// TIA Portal project "1905391_000_002" (V16)

(* hardware
DEVICE "S7-1200 station_1"  S7-1200 Station
   slot 0: "Rack_0"  S7-1200 Rack  Rack  V1.0
   slot 1: "PLC_1"  CPU 1211C DC/DC/DC  6ES7 211-1AE40-0XB0  V4.4
DEVICE "HMI_1"  TP900 Comfort
   slot 0: "HMI_1"  TP900 Comfort  6AV2 124-0JC01-0AX0  16.0.0.0
   slot 1: "HMI_RT_1"  TP900 Comfort  6AV2 124-0JC01-0AX0  16.0.0.0
   slot 5: "HMI_1.IE_CP_1"  PROFINET Interface  16.0.0.0
      slot 1: "PROFINET Interface_1"  PROFINET Interface
         slot 1: "Port_1"  Port
         slot 2: "Port_2"  Port
   slot 7: "HMI_1.MPI/DP_CP_1"  MPI/DP Interface  16.0.0.0
*)

// ===== PLC "PLC_1"  CPU 1211C DC/DC/DC =====

VAR_GLOBAL   // PLC tag table "Default tag table"
   "System_Byte" AT %MB1 : Byte;
   "FirstScan" AT %M1.0 : Bool;
   "DiagStatusUpdate" AT %M1.1 : Bool;
   "AlwaysTRUE" AT %M1.2 : Bool;
   "AlwaysFALSE" AT %M1.3 : Bool;
   "Clock_Byte" AT %MB0 : Byte;
   "Clock_10Hz" AT %M0.0 : Bool;
   "Clock_5Hz" AT %M0.1 : Bool;
   "Clock_2.5Hz" AT %M0.2 : Bool;
   "Clock_2Hz" AT %M0.3 : Bool;
   "Clock_1.25Hz" AT %M0.4 : Bool;
   "Clock_1Hz" AT %M0.5 : Bool;
   "Clock_0.625Hz" AT %M0.6 : Bool;
   "Clock_0.5Hz" AT %M0.7 : Bool;
END_VAR

VAR_GLOBAL CONSTANT   // PLC tag table "Default tag table"
   "STRING_LENGTH" : Int := 20;
   "ADP_PARAMETER_LENGTH" : Int := 5;
END_VAR

TYPE "Database.UDT"
   STRUCT
      elements : "Elements.Data.UDT";
      wires : "Wires.Data.UDT";
   END_STRUCT;
END_TYPE

TYPE "Row.(IOF.String_IOF.String).UDT"
   STRUCT
      cell_00 : "IO_Field.String.UDT";
      cell_01 : "IO_Field.String.UDT";
   END_STRUCT;
END_TYPE

TYPE "IO_Field.String.UDT"
   STRUCT
      animation : Int;
      enable : Bool;
      input_finished : Bool;
      visible : Bool;
      value : String["STRING_LENGTH"];
   END_STRUCT;
END_TYPE

TYPE "HMI_Interface.UDT"
   STRUCT
      elements : "Elements.HMI.UDT";
      wires : "Wires.HMI.UDT";
   END_STRUCT;
END_TYPE

TYPE "LED_Interface.UDT"
   STRUCT
      elements : "Elements.LED.UDT";
      wires : "Wires.LED.UDT";
   END_STRUCT;
END_TYPE

TYPE "Row.(IOF.String_IOF.Real).UDT"
   STRUCT
      cell_00 : "IO_Field.String.UDT";
      cell_01 : "IO_Field.Real.UDT";
   END_STRUCT;
END_TYPE

TYPE "IO_Field.Real.UDT"
   STRUCT
      animation : Int;
      enable : Bool;
      input_finished : Bool;
      visible : Bool;
      value : Real;
   END_STRUCT;
END_TYPE

// folder: ADP Data

TYPE "ADP.Row.2_Cells.UDT"
   STRUCT
      me : Array[0..1] of "ADP.Cell.UDT";
   END_STRUCT;
END_TYPE

TYPE "ADP.Cell.UDT"
   STRUCT
      color : String["ADP_PARAMETER_LENGTH"];
      flashing : String["ADP_PARAMETER_LENGTH"];
      h_align : String["ADP_PARAMETER_LENGTH"];
      lince_control : String["ADP_PARAMETER_LENGTH"];
      scroll_speed : String["ADP_PARAMETER_LENGTH"];
      size_and_face : String["ADP_PARAMETER_LENGTH"];
      v_align : String["ADP_PARAMETER_LENGTH"];
      value : String["STRING_LENGTH"];
   END_STRUCT;
END_TYPE

TYPE "ADP.Message_Buffer.UDT"
   STRUCT
      me : Array[0..999] of Byte;
   END_STRUCT;
END_TYPE

TYPE "ADP.Decoded.UDT"
   STRUCT
      color : "ADP.Decoded.Color.UDT";
      flash : "ADP.Decoded.Flash.UDT";
      horizontal_alignment : "ADP.Decoded.Horizontal_Alignment.UDT";
      line_control : "ADP.Decoded.Line_Control.UDT";
      scroll_speed : "ADP.Decoded.Scroll_Speed.UDT";
      size_and_face : "ADP.Decoded.Size_and_Face.UDT";
      vertical_alignment : "ADP.Decoded.Vertical_Alignment.UDT";
   END_STRUCT;
END_TYPE

TYPE "ADP.Decoded.Color.UDT"
   STRUCT
      black : String[8] := 'black';
      blue : String[8] := 'blue';
      green : String[8] := 'green';
      mix_1 : String[8] := 'mix 1';
      mix_2 : String[8] := 'mix 2';
      mix_3 : String[8] := 'mix 3';
      mix_4 : String[8] := 'mix 4';
      red : String[8] := 'red';
      white : String[8] := 'white';
      yellow : String[8] := 'yellow';
   END_STRUCT;
END_TYPE

TYPE "ADP.Decoded.Flash.UDT"
   STRUCT
      off : String[8] := 'off';
      on : String[8] := 'on';
   END_STRUCT;
END_TYPE

TYPE "ADP.Decoded.Horizontal_Alignment.UDT"
   STRUCT
      center : String[8] := 'center';
      left : String[8] := 'left';
      right : String[8] := 'right';
   END_STRUCT;
END_TYPE

TYPE "ADP.Encoded.UDT"
VERSION : 0.1
   STRUCT
      file_system : "ADP.Encoded.File_System.UDT";
      formatting : "ADP.Encoded.Formatting.UDT";
   END_STRUCT;
END_TYPE

TYPE "ADP.Message_Formats.Encoded.UDT"
   STRUCT
      color : String [5];
      flash : String [5];
      scroll_speed : String [5];
      size_and_face : String [5];
      vertical_alignment : String [5];
      horizontal_alignment : String [5];
   END_STRUCT;
END_TYPE

TYPE "ADP.Message_Formats.Decoded.UDT"
   STRUCT
      color : String [20];
      flash : String [20];
      scroll_speed : String [20];
      size_and_face : String [20];
      vertical_alignment : String [20];
      horizontal_alignment : String [20];
   END_STRUCT;
END_TYPE

TYPE "ADP.Decoded.Scroll_Speed.UDT"
   STRUCT
      slowest : String[9] := 'slowest';
      slow : String[9] := 'slow';
      normal : String[9] := 'normal';
      fast : String[9] := 'fast';
      fastest : String[9] := 'fastest';
   END_STRUCT;
END_TYPE

TYPE "ADP.Decoded.Size_and_Face.UDT"
   STRUCT
      bold_5 : String[11] := 'bold 5';
      bold_11 : String[11] := 'bold 11';
      bold_14 : String[11] := 'bold 14';
      bold_15 : String[11] := 'bold 15';
      bold_16 : String[11] := 'bold 16';
      bold_22 : String[11] := 'bold 22';
      bold_30 : String[11] := 'bold 30';
      bold_32 : String[11] := 'bold 32';
      bold_40 : String[11] := 'bold 40';
      normal_5 : String[11] := 'normal 5';
      normal_7 : String[11] := 'normal 7';
      normal_9 : String[11] := 'normal 9';
      normal_11 : String[11] := 'normal 11';
      normal_14 : String[11] := 'normal 14';
      normal_15 : String[11] := 'normal 15';
      normal_16 : String[11] := 'normal 16';
      normal_22 : String[11] := 'normal 22';
      normal_24 : String[11] := 'normal 24';
      normal_30 : String[11] := 'normal 30';
      normal_32 : String[11] := 'normal 32';
      normal_40 : String[11] := 'normal 40';
   END_STRUCT;
END_TYPE

TYPE "ADP.Decoded.Vertical_Alignment.UDT"
   STRUCT
      bottom_hold : String[15] := 'bottom hold';
      fill_hold : String[15] := 'fill hold';
      middle_hold : String[15] := 'middle hold';
      top_hold : String[15] := 'top hold';
      bottom_scroll : String[15] := 'bottom scroll';
      fill_scroll : String[15] := 'fill scroll';
      middle_scroll : String[15] := 'middle scroll';
      top_scroll : String[15] := 'top scroll';
   END_STRUCT;
END_TYPE

TYPE "ADP.Encoded.File_System.UDT"
   STRUCT
      "00 Start of Header" : String[5] := '$01';
      "01 Address" : String[5] := 'Z00';
      "02 Start of Text" : String[5] := '$02';
      "03 Command & File" : String[5] := 'AA';
      "04 END" : String[5] := '$04';
   END_STRUCT;
END_TYPE

TYPE "ADP.Encoded.Formatting.UDT"
   STRUCT
      color : "ADP.Encoded.Formatting.Color.UDT";
      flashing : "ADP.Encoded.Formatting.Flashing.UDT";
      horizontal_alignment : "ADP.Encoded.Formatting.Horizonta_Alignment.UDT";
      line_control : "ADP.Encoded.Formatting.Line_Control.UDT";
      scroll_speed : "ADP.Encoded.Formatting.Scroll_Speed.UDT";
      size_and_face : "ADP.Encoded.Formatting.Size_and_Face.UDT";
      vertical_alignment : "ADP.Encoded.Formatting.Vertical_Alignment.UDT";
   END_STRUCT;
END_TYPE

TYPE "ADP.Encoded.Formatting.Color.UDT"
   STRUCT
      black : String[5] := '$1C0';
      blue : String[5] := '$1C8';
      green : String[5] := '$1C2';
      mix_1 : String[5] := '$1C4';
      mix_2 : String[5] := '$1C5';
      mix_3 : String[5] := '$1C6';
      mix_4 : String[5] := '$1CY';
      red : String[5] := '$1C1';
      white : String[5] := '$1C9';
      yellow : String[5] := '$1C3';
   END_STRUCT;
END_TYPE

TYPE "ADP.Encoded.Formatting.Flashing.UDT"
   STRUCT
      off : String[5] := '$070';
      on : String[5] := '$071';
   END_STRUCT;
END_TYPE

TYPE "ADP.Encoded.Formatting.Size_and_Face.UDT"
   STRUCT
      bold_5 : String[5] := '$1AG';
      bold_11 : String[5] := '$1AH';
      bold_14 : String[5] := '$1A5';
      bold_15 : String[5] := '$1A6';
      bold_16 : String[5] := '$1A7';
      bold_22 : String[5] := '$1AC';
      bold_30 : String[5] := '$1AI';
      bold_32 : String[5] := '$1AJ';
      bold_40 : String[5] := '$1AK';
      normal_5 : String[5] := '$1A0';
      normal_7 : String[5] := '$1A1';
      normal_9 : String[5] := '$1A8';
      normal_11 : String[5] := '$1A9';
      normal_14 : String[5] := '$1A2';
      normal_15 : String[5] := '$1A3';
      normal_16 : String[5] := '$1A4';
      normal_22 : String[5] := '$1AA';
      normal_24 : String[5] := '$1AB';
      normal_30 : String[5] := '$1AD';
      normal_32 : String[5] := '$1AE';
      normal_40 : String[5] := '$1AF';
   END_STRUCT;
END_TYPE

TYPE "ADP.Encoded.Formatting.Horizonta_Alignment.UDT"
   STRUCT
      center : String[5] := '$L1';
      left : String[5] := '$L0';
      right : String[5] := '$L2';
   END_STRUCT;
END_TYPE

TYPE "ADP.Encoded.Formatting.Vertical_Alignment.UDT"
   STRUCT
      middle_hold : String[5] := '$1B b';
      fill_hold : String[5] := '$1B"b';
      bottom_hold : String[5] := '$1B&b';
      top_hold : String[5] := '$1B0b';
      bottom_scroll : String[5] := '$1B a';
      fill_scroll : String[5] := '$1B"a';
      middle_scroll : String[5] := '$1B&a';
      top_scroll : String[5] := '$1B0a';
   END_STRUCT;
END_TYPE

TYPE "ADP.Encoded.Formatting.Scroll_Speed.UDT"
   STRUCT
      slowest : String[5] := '$15';
      slow : String[5] := '$16';
      normal : String[5] := '$17';
      fast : String[5] := '$18';
      fastest : String[5] := '$19';
   END_STRUCT;
END_TYPE

TYPE "ADP.Encoded.Formatting.Line_Control.UDT"
   STRUCT
      new_line : String[5] := '$R';
      word_wrap : String[5] := '';
   END_STRUCT;
END_TYPE

TYPE "ADP.Decoded.Line_Control.UDT"
   STRUCT
      new_line : String[9] := 'new line';
      word_wrap : String[9] := 'word wrap';
   END_STRUCT;
END_TYPE

// folder: Element Data

TYPE "Elements.HMI.UDT"
   STRUCT
      chromium : "Row.(IOF.String_IOF.Real).UDT";
      custom : "Row.(IOF.String_IOF.Real).UDT";
      header : "Row.(IOF.String_IOF.String).UDT";
      heat : "Row.(IOF.String_IOF.Real).UDT";
      manganese : "Row.(IOF.String_IOF.Real).UDT";
      molybdenum : "Row.(IOF.String_IOF.Real).UDT";
      nickel : "Row.(IOF.String_IOF.Real).UDT";
      silicon : "Row.(IOF.String_IOF.Real).UDT";
      vanadium : "Row.(IOF.String_IOF.Real).UDT";
   END_STRUCT;
   // header.cell_00.value := 'Material';
   // header.cell_01.value := 'Bags';
END_TYPE

TYPE "Elements.Data.UDT"
   STRUCT
      chromium : Real;
      custom : Real;
      heat : Real;
      manganese : Real;
      molybdenum : Real;
      nickel : Real;
      silicon : Real;
      vanadium : Real;
   END_STRUCT;
END_TYPE

TYPE "Elements.LED.UDT"
   STRUCT
      chromium : "ADP.Row.2_Cells.UDT";
      custom : "ADP.Row.2_Cells.UDT";
      header : "ADP.Row.2_Cells.UDT";
      heat : "ADP.Row.2_Cells.UDT";
      manganese : "ADP.Row.2_Cells.UDT";
      molybdenum : "ADP.Row.2_Cells.UDT";
      nickel : "ADP.Row.2_Cells.UDT";
      silicon : "ADP.Row.2_Cells.UDT";
      vanadium : "ADP.Row.2_Cells.UDT";
   END_STRUCT;
   // chromium.me[0].value := 'chromium';
   // heat.me[0].value := 'heat';
   // manganese.me[0].value := 'manganese';
   // molybdenum.me[0].value := 'molybdenum';
   // nickel.me[0].value := 'nickel';
   // silicon.me[0].value := 'silicon';
   // vanadium.me[0].value := 'vanadium';
   // custom.me[0].value := 'Custom';
   // header.me[0].value := 'Material';
   // header.me[1].value := 'Bags';
END_TYPE

// folder: Wire Data

TYPE "Wires.Data.UDT"
   STRUCT
      aluminum : Real;
      calcium_silicon : Real;
      carbon : Real;
      custom : Real;
      heat : Real;
      sulfur : Real;
   END_STRUCT;
END_TYPE

TYPE "Wires.LED.UDT"
   STRUCT
      aluminum : "ADP.Row.2_Cells.UDT";
      calcium_silicon : "ADP.Row.2_Cells.UDT";
      carbon : "ADP.Row.2_Cells.UDT";
      custom : "ADP.Row.2_Cells.UDT";
      heat : "ADP.Row.2_Cells.UDT";
      sulfur : "ADP.Row.2_Cells.UDT";
   END_STRUCT;
   // aluminum.me[0].value := 'AL Wire';
   // calcium_silicon.me[0].value := 'Cal/Sil Wire';
   // carbon.me[0].value := 'Carbon Wire';
   // heat.me[0].value := 'HEAT';
   // sulfur.me[0].value := 'Sulfur Wire';
   // custom.me[0].value := 'Custom';
END_TYPE

TYPE "Wires.HMI.UDT"
   STRUCT
      aluminum : "Row.(IOF.String_IOF.Real).UDT";
      calcium_silicon : "Row.(IOF.String_IOF.Real).UDT";
      carbon : "Row.(IOF.String_IOF.Real).UDT";
      custom : "Row.(IOF.String_IOF.Real).UDT";
      header : "Row.(IOF.String_IOF.String).UDT";
      heat : "Row.(IOF.String_IOF.Real).UDT";
      sulfur : "Row.(IOF.String_IOF.Real).UDT";
   END_STRUCT;
   // header.cell_00.value := 'Material';
   // header.cell_01.value := 'Feet';
END_TYPE

// folder: data

DATA_BLOCK "Database.Data"   // DB1
{ S7_Optimized_Access := 'TRUE' }
VERSION : 0.1
BEGIN
END_DATA_BLOCK

// folder: display/HMI

DATA_BLOCK "HMI_Interface.Data"   // DB2
{ S7_Optimized_Access := 'TRUE' }
VERSION : 0.1
BEGIN
END_DATA_BLOCK

// folder: display/LED

DATA_BLOCK "LED_Interface.Data"   // DB3
{ S7_Optimized_Access := 'TRUE' }
VERSION : 0.1
BEGIN
END_DATA_BLOCK

// folder: (top level)

FUNCTION "Strip_Sign" : String   // FC20, SCL
{ S7_Optimized_Access := 'TRUE' }
VERSION : 0.1
   VAR_INPUT
      "string" : String;
   END_VAR
   VAR_TEMP
      Length : Int;
      "String Box" : String;
      "Test Character" : String;
   END_VAR
   VAR CONSTANT
      "+" : Char := '+';
      "-" : Char := '-';
   END_VAR
BEGIN
   #"String Box" := #string;
   #"Test Character" := LEFT_STRING(IN := #"String Box",
                                    L := 1);
   IF #"Test Character" = #"+" OR #"Test Character" = #"-" THEN
       #Length := LEN(#"String Box");
       #"String Box" := RIGHT_STRING(IN := #"String Box", L := #Length - 1);

   END_IF;
   #"Strip Sign" := #"String Box";
END_FUNCTION

FUNCTION "Trim" : String   // FC21, SCL
{ S7_Optimized_Access := 'TRUE' }
AUTHOR : Machado
FAMILY : String
VERSION : 1.0
// removes leading and trailing whitespace from input string
   VAR_INPUT
      "string" : String;
   END_VAR
   VAR_TEMP
      ret : String;
   END_VAR
   VAR CONSTANT
      space : String := ' ';
   END_VAR
BEGIN
   #ret := #string;
   WHILE LEFT(IN := #ret, L := 1) = #space DO
       #ret := RIGHT(IN := #ret, L := LEN(#ret) - 1);
   END_WHILE;
   WHILE RIGHT(IN := #ret, L := 1) = #space DO
       #ret := LEFT(IN := #ret, L := LEN(#ret) - 1);
   END_WHILE;
   #Trim := #ret;
END_FUNCTION

FUNCTION "Upper" : String   // FC22, SCL
{ S7_Optimized_Access := 'TRUE' }
AUTHOR : Machado
FAMILY : String
VERSION : 1.0
// returns the input string converted to all upper case
   VAR_INPUT
      "string" : String;
   END_VAR
   VAR_TEMP
      "type" : Bool;
      stringBox : String;
      status : Int;
      charArr : Array[0..255] of Char;
      cntChar : UInt;
      pChar : Int;
   END_VAR
   VAR CONSTANT
      asciiLow : Char := 'a';
      asciiHigh : Char := 'z';
      asciiCaseOffset : Int := 32;
   END_VAR
BEGIN
   Strg_TO_Chars(Strg := #string,
                 pChars := 0,
                 Cnt => #cntChar,
                 Chars := #charArr);

   FOR #pChar := 0 TO UINT_TO_INT(#cntChar) - 1 DO
       IF #asciiLow <= #charArr[#pChar] AND #charArr[#pChar] <= #asciiHigh THEN
           #charArr[#pChar] := INT_TO_CHAR(CHAR_TO_INT(#charArr[#pChar]) - #asciiCaseOffset);
       END_IF;
   END_FOR;

   Chars_TO_Strg(Chars := #charArr,
                 pChars := 0,
                 Cnt := #cntChar,
                 Strg => #stringBox);

   #Upper := #stringBox;
END_FUNCTION

ORGANIZATION_BLOCK "Main"   // OB1, LAD, ProgramCycle
TITLE = "Main Program Sweep (Cycle)"
{ S7_Optimized_Access := 'TRUE' }
VERSION : 0.1
   VAR_INPUT
      Initial_Call : Bool;   // Initial call of this OB
      Remanence : Bool;   // =True, if remanent data are available
   END_VAR
BEGIN
END_ORGANIZATION_BLOCK

// folder: display

FUNCTION_BLOCK "Display"   // FB5, SCL
{ S7_Optimized_Access := 'TRUE' }
VERSION : 0.1
BEGIN
   REGION "HMI"

   END_REGION

   REGION "LED"

   END_REGION
END_FUNCTION_BLOCK

// folder: display/HMI

FUNCTION_BLOCK "HMI"   // FB6, SCL
{ S7_Optimized_Access := 'TRUE' }
VERSION : 0.1
   VAR_IN_OUT
      interface : "HMI_Interface.UDT";
   END_VAR
   VAR
      place_holder : Bool;
   END_VAR
BEGIN
   REGION "VALIDATE INPUT"
       "HMI.Validate"();
   END_REGION


   REGION "DISPLAY VALUES"
       // may not be needed, handeled entirely in middleware
   END_REGION


   REGION "ANIMATE"
       "HMI.Animate"();
   END_REGION
END_FUNCTION_BLOCK

FUNCTION "HMI.Animate" : Void   // FC8, SCL
{ S7_Optimized_Access := 'TRUE' }
VERSION : 0.1
BEGIN
   "Element.Animate"();
   "Wire.Animate"();
END_FUNCTION

FUNCTION "HMI.Validate" : Void   // FC9, SCL
{ S7_Optimized_Access := 'TRUE' }
VERSION : 0.1
BEGIN
   "Element.Validate"();
   "Wire.Validate"();
END_FUNCTION

FUNCTION "HMI.Display" : Void   // FC10, SCL
{ S7_Optimized_Access := 'TRUE' }
VERSION : 0.1
   VAR_INPUT
      database : Bool;
   END_VAR
BEGIN
END_FUNCTION

// folder: display/LED

FUNCTION_BLOCK "LED"   // FB7, SCL
{ S7_Optimized_Access := 'TRUE' }
VERSION : 0.1
   VAR
      Elements_Sign : "Elements_Sign";
      Wires_Sign : "Wires_Sign";
   END_VAR
BEGIN
   REGION "ELEMENTS"
       #Elements_Sign();
   END_REGION

   REGION "WIRES"
       #Wires_Sign();
   END_REGION
END_FUNCTION_BLOCK

FUNCTION_BLOCK "LED.Sign.Send"   // FB9, SCL
{ S7_Optimized_Access := 'TRUE' }
VERSION : 0.1
   VAR_INPUT
      data : "ADP.Message_Buffer.UDT";
      id : Conn_Ouc;
      request : Bool;
   END_VAR
   VAR
      TSEND : TSEND;
   END_VAR
BEGIN
   #TSEND(REQ := #request,
          ID := #id,
          DATA := #data);
END_FUNCTION_BLOCK

FUNCTION_BLOCK "LED.Sign"   // FB10, SCL
{ S7_Optimized_Access := 'TRUE' }
VERSION : 0.1
   VAR_INPUT
      id : Conn_Ouc;
      connection_parameters : TCON_Param;
      requests : Struct
         connect : Bool;
         diagnostics : Bool;
         disconnect : Bool;
         reset : Bool;
         send : Bool;
      END_STRUCT;
   END_VAR
   VAR
      Connect : "LED.Sign.Connect";
      Disconnect : "LED.Sign.Disconnect";
      Send : "LED.Sign.Send";
      Reset : "LED.Sign.Reset";
      Diagnostics : "LED.Sign.Diagnostics";
   END_VAR
BEGIN
   #Connect(request := #requests.connect,
            id := #id,
            connection_parameters := #connection_parameters);

   #Disconnect(id := #id,
               request := #requests.disconnect);

   #Send(id := #id,
         request := #requests.send);

   #Reset(id := #id,
          request := #requests.reset);

   #Diagnostics(id := #id,
                request := #requests.diagnostics);
END_FUNCTION_BLOCK

FUNCTION_BLOCK "LED.Sign.Connect"   // FB11, SCL
{ S7_Optimized_Access := 'TRUE' }
VERSION : 0.1
   VAR_INPUT
      request : Bool;
      id : Conn_Ouc;
      connection_parameters : TCON_Param;
   END_VAR
   VAR
      TCON : TCON;
   END_VAR
BEGIN
   #TCON(REQ := #request,
         ID := #id,
         CONNECT := #connection_parameters);
END_FUNCTION_BLOCK

FUNCTION_BLOCK "LED.Sign.Reset"   // FB12, SCL
{ S7_Optimized_Access := 'TRUE' }
VERSION : 0.1
   VAR_INPUT
      request : Bool;
      id : Conn_Ouc;
   END_VAR
   VAR
      T_RESET : T_RESET;
   END_VAR
BEGIN
   #T_RESET(REQ:=#request,
            ID:=#id,
            DONE=>_bool_out_,
            BUSY=>_bool_out_,
            ERROR=>_bool_out_,
            STATUS=>_word_out_);
END_FUNCTION_BLOCK

FUNCTION_BLOCK "LED.Sign.Disconnect"   // FB13, SCL
{ S7_Optimized_Access := 'TRUE' }
VERSION : 0.1
   VAR_INPUT
      request : Bool;
      id : Conn_Ouc;
   END_VAR
   VAR
      TDISCON : TDISCON;
   END_VAR
BEGIN
   #TDISCON(REQ := #request,
            ID := #id);
END_FUNCTION_BLOCK

FUNCTION_BLOCK "LED.Sign.Diagnostics"   // FB14, SCL
{ S7_Optimized_Access := 'TRUE' }
VERSION : 0.1
   VAR_INPUT
      request : Bool;
      id : Conn_Ouc;
   END_VAR
   VAR
      T_DIAG : T_DIAG;
   END_VAR
BEGIN
   #T_DIAG(REQ:=#request,
           ID:=#id);
END_FUNCTION_BLOCK

// folder: display/LED/Elements Sign

FUNCTION_BLOCK "Elements_Sign"   // FB16, SCL
{ S7_Optimized_Access := 'TRUE' }
VERSION : 0.1
   VAR
      Sign : "LED.Sign";
      id : Conn_Ouc;
      connection_parameters : TCON_Param;
   END_VAR
BEGIN
   "Elements_Sign.Assemble_Message"();
   #Sign(id := #id,
         connection_parameters := #connection_parameters);
END_FUNCTION_BLOCK

FUNCTION "Elements_Sign.Assemble_Message" : Void   // FC11, SCL
{ S7_Optimized_Access := 'TRUE' }
VERSION : 0.1
BEGIN
END_FUNCTION

// folder: display/LED/Wires Sign

FUNCTION_BLOCK "Wires_Sign"   // FB15, SCL
{ S7_Optimized_Access := 'TRUE' }
VERSION : 0.1
   VAR
      Sign : "LED.Sign";
      id : Conn_Ouc;
      connection_parameters : TCON_Param;
   END_VAR
BEGIN
   "Wires_Sign.Assemble_Message"();
   #Sign(id := #id,
         connection_parameters := #connection_parameters);
END_FUNCTION_BLOCK

FUNCTION "Wires_Sign.Assemble_Message" : Void   // FC12, SCL
{ S7_Optimized_Access := 'TRUE' }
VERSION : 0.1
BEGIN
END_FUNCTION

// folder: element

FUNCTION_BLOCK "Elements"   // FB3, SCL
{ S7_Optimized_Access := 'TRUE' }
VERSION : 0.1
   VAR_IN_OUT
      database : "Elements.Data.UDT";
      hmi : "Elements.HMI.UDT";
      led : "Elements.LED.UDT";
   END_VAR
   VAR
      Chromium : "Element";
      Custom : "Element";
      Heat : "Element";
      Manganese : "Element";
      Molybdenum : "Element";
      Nickel : "Element";
      Silicon : "Element";
      Vanadium : "Element";
   END_VAR
BEGIN
   #Chromium(database := #database.chromium,
             hmi := #hmi.chromium,
             led := #led.chromium);

   #Custom(database := #database.custom,
           hmi := #hmi.custom,
           led := #led.custom);

   #Heat(database := #database.heat,
         hmi := #hmi.heat,
         led := #led.heat);

   #Manganese(database := #database.manganese,
              hmi := #hmi.manganese,
              led := #led.manganese);

   #Molybdenum(database := #database.molybdenum,
               hmi := #hmi.molybdenum,
               led := #led.molybdenum);    

   #Nickel(database := #database.nickel,
           hmi := #hmi.nickel,
           led := #led.nickel);

   #Silicon(database := #database.silicon,
            hmi := #hmi.silicon,
            led := #led.silicon);

   #Vanadium(database := #database.vanadium,
             hmi := #hmi.vanadium,
             led := #led.vanadium);
END_FUNCTION_BLOCK

FUNCTION_BLOCK "Element"   // FB8, SCL
{ S7_Optimized_Access := 'TRUE' }
VERSION : 0.1
   VAR_IN_OUT
      database : Real;
      hmi : "Row.(IOF.String_IOF.Real).UDT";
      led : "ADP.Row.2_Cells.UDT";
   END_VAR
BEGIN
   REGION "READ"
       "Element.Read"(database := #database,
                      hmi := #hmi,
                      led := #led);
   END_REGION


   REGION "WRITE"
       IF #hmi.cell_01.input_finished THEN
           #hmi.cell_01.input_finished := FALSE;
           #database := "Element.Set"(#hmi.cell_01.value);
       END_IF;
   END_REGION
END_FUNCTION_BLOCK

FUNCTION "Element.Validate" : Void   // FC4, SCL
{ S7_Optimized_Access := 'TRUE' }
VERSION : 0.1
   VAR_IN_OUT
      hmi : "Row.(IOF.String_IOF.Real).UDT";
   END_VAR
   VAR_TEMP
      _validation : Bool;
   END_VAR
BEGIN
   // currently no validation conditons
   #_validation := TRUE;
   "Material.Validate"(valid := #_validation,
                       hmi := #hmi);
END_FUNCTION

FUNCTION "Element.Animate" : Void   // FC6, SCL
{ S7_Optimized_Access := 'TRUE' }
VERSION : 0.1
   VAR_IN_OUT
      row : "Row.(IOF.String_IOF.Real).UDT";
   END_VAR
BEGIN
   "Material.Animate"(#row);
END_FUNCTION

FUNCTION "Element.Set" : Real   // FC13, SCL
{ S7_Optimized_Access := 'TRUE' }
VERSION : 0.1
   VAR_INPUT
      hmi : "Row.(IOF.String_IOF.Real).UDT";
   END_VAR
   VAR_IN_OUT
      database : Real;
   END_VAR
BEGIN
   "Material.Set"(hmi := #hmi,
                  database := #database);
END_FUNCTION

FUNCTION "Element.Read.HMI" : Void   // FC14, SCL
{ S7_Optimized_Access := 'TRUE' }
VERSION : 0.1
   VAR_INPUT
      database : Real;
   END_VAR
   VAR_IN_OUT
      hmi : "Row.(IOF.String_IOF.Real).UDT";
   END_VAR
BEGIN
   "Material.Read.HMI"(database := #database,
                       hmi := #hmi);
END_FUNCTION

FUNCTION "Element.Read" : Void   // FC15, SCL
{ S7_Optimized_Access := 'TRUE' }
VERSION : 0.1
   VAR_INPUT
      database : Real;
   END_VAR
   VAR_IN_OUT
      hmi : "Row.(IOF.String_IOF.Real).UDT";
      led : "ADP.Row.2_Cells.UDT";
   END_VAR
BEGIN
   "Element.Read.HMI"(database := #database,
                      hmi := #hmi);

   "Element.Read.LED"(database := #database,
                      led := #led);
END_FUNCTION

FUNCTION "Element.Read.LED" : Void   // FC18, SCL
{ S7_Optimized_Access := 'TRUE' }
VERSION : 0.1
   VAR_INPUT
      database : Real;
   END_VAR
   VAR_IN_OUT
      led : "ADP.Row.2_Cells.UDT";
   END_VAR
BEGIN
   "Material.Read.LED"(database := #database,
                       led := #led);
END_FUNCTION

FUNCTION "Element.Scale" : Real   // FC19, SCL
{ S7_Optimized_Access := 'TRUE' }
VERSION : 0.1
   VAR_INPUT
      value : Real;
   END_VAR
BEGIN
   #"Element.Scale" := "Material.Scale"(#value);
END_FUNCTION

// folder: material

FUNCTION "Material.Read.HMI" : Void   // FC23, SCL
{ S7_Optimized_Access := 'TRUE' }
VERSION : 0.1
   VAR_INPUT
      database : Real;
   END_VAR
   VAR_IN_OUT
      hmi : "Row.(IOF.String_IOF.Real).UDT";
   END_VAR
BEGIN
   #hmi.cell_01.value := #database;
END_FUNCTION

FUNCTION "Material.Set" : Void   // FC23, SCL
{ S7_Optimized_Access := 'TRUE' }
VERSION : 0.1
   VAR_INPUT
      hmi : "Row.(IOF.String_IOF.Real).UDT";
   END_VAR
   VAR_IN_OUT
      database : Real;
   END_VAR
BEGIN
   #database :=  "Material.Scale"(#hmi.cell_01.value);
END_FUNCTION

FUNCTION "Material.Validate" : Void   // FC23, SCL
{ S7_Optimized_Access := 'TRUE' }
VERSION : 0.1
   VAR_INPUT
      valid : Bool;
   END_VAR
   VAR_IN_OUT
      hmi : "Row.(IOF.String_IOF.Real).UDT";
   END_VAR
BEGIN
   REGION "NOTES"
       (*
           Validation conditions go in child.
           Results passed as simple bool.
           Process:
               1. check hmi value
               2. if value is acceptable do nothing
               3. if value is unacceptable:
                   a. clear hmi value
                   b. reset input_finished to prevent middleware
                      from writing value to database
       *)
   END_REGION

   REGION "INVALID"
       IF #valid THEN
           #hmi.cell_01.value := 0.0;
           #hmi.cell_01.input_finished := FALSE;
           RETURN;
       END_IF;
   END_REGION

   REGION "VALID"
       // DO NOTHING
       RETURN;
   END_REGION
END_FUNCTION

FUNCTION "Material.Scale" : Real   // FC23, SCL
{ S7_Optimized_Access := 'TRUE' }
VERSION : 0.1
   VAR_INPUT
      value : Real;
   END_VAR
BEGIN
   #"Material.Scale" := #value;
END_FUNCTION

FUNCTION "Material.Read.LED" : Void   // FC23, SCL
{ S7_Optimized_Access := 'TRUE' }
VERSION : 0.1
   VAR_INPUT
      database : Real;
   END_VAR
   VAR_IN_OUT
      led : "ADP.Row.2_Cells.UDT";
   END_VAR
BEGIN
   #led.me[1].value := "Trim"("Strip_Sign"(REAL_TO_STRING(#database)));
END_FUNCTION

FUNCTION "Material.Animate" : Void   // FC24, SCL
{ S7_Optimized_Access := 'TRUE' }
VERSION : 0.1
   VAR_IN_OUT
      row : Variant;
   END_VAR
   VAR_TEMP
      _symbol_name : String;
      _real_row : "Row.(IOF.String_IOF.Real).UDT";
      _status : Int;
      _string_row : "Row.(IOF.String_IOF.Real).UDT";
   END_VAR
   VAR CONSTANT
      BLACK_BLACK : Int := 0;
      WHITE_BACKGROUND : Int := 1;
      WHITE_FOREGROUND : Int := 2;
      WHITE_FLASHING : Int := 3;
      GRAY_BACKGROUND : Int := 4;
      GRAY_FOREGROUND : Int := 5;
      GRAY_FLASHING : Int := 6;
      RED_LIGHT_BACKGROUND : Int := 7;
      RED_LIGTH_FOREGROUND : Int := 8;
      RED_LIGHT_FLASHING : Int := 9;
      RED_BACKGROUND : Int := 10;
      RED_FOREGROUND : Int := 11;
      RED_FLASHING : Int := 12;
      YELLOW_LIGHT_BACKGROUND : Int := 13;
      YELLOW_LIGHT_FOREGROUND : Int := 14;
      YELLOW_LIGHT_FLASHING : Int := 15;
      YELLOW_BACKGROUND : Int := 16;
      YELLOW_FOREGROUND : Int := 17;
      YELLOW_FLASHING : Int := 18;
      GREEN_LIGHT_BACKGROUND : Int := 19;
      GREEN_LIGHT_FOREGROUND : Int := 20;
      GREEN_LIGHT_FLASHING : Int := 21;
      GREEN_BACKGROUND : Int := 22;
      GREEN_FOREGROUND : Int := 23;
      GREEN_FLASHING : Int := 24;
      TEAL_LIGHT_BACKGROUND : Int := 25;
      TEAL_LIGHT_FOREGROUND : Int := 26;
      TEAL_LIGHT_FLASHING : Int := 27;
      TEAL_BACKGROUND : Int := 28;
      TEAL_FOREGROUND : Int := 29;
      TEAL_FLASHING : Int := 30;
      BLUE_LIGHT_BACKGROUND : Int := 31;
      BLUE_LIGHT_FOREGROUND : Int := 32;
      BLUE_LIGHT_FLASHING : Int := 33;
      BLUE_BACKGROUND : Int := 34;
      BLUE_FOREGROUND : Int := 35;
      BLUE_FLASHING : Int := 36;
      PURPLE_LIGHT_BACKGROUND : Int := 37;
      PURPLE_LIGHT_FOREGROUND : Int := 38;
      PURPLE_LIGHT_FLASHING : Int := 39;
      PURPLE_DARK_BACKGROUND : Int := 40;
      PURPLE_DARK_FOREGROUND : Int := 41;
      PURPLE_FLASHING : Int := 42;
      DISABLED : Int := 254;
      INVISIBLE : Int := 255;
      LBlDRd : Int := 43;
      DRdLBl : Int := 44;
      LBlDRdFl : Int := 45;
      DBlDRd : Int := 46;
      DRdDBl : Int := 47;
      DBlDRdFl : Int := 48;
   END_VAR
BEGIN
   #_symbol_name := WSTRING_TO_STRING(GetSymbolName(variable := #row, size := 0));

   IF FIND(IN1 := #_symbol_name, IN2 := 'header') = 0 THEN
       #_status := MOVE_BLK_VARIANT(SRC := #row,
                                    COUNT := 1,
                                    SRC_INDEX := 0,
                                    DEST_INDEX := 0,
                                    DEST => #_real_row);
       #_real_row.cell_00.animation := #GRAY_BACKGROUND;
       #_real_row.cell_01.animation := #WHITE_BACKGROUND;
       #_status := MOVE_BLK_VARIANT(SRC := #_real_row,
                                    COUNT := 1,
                                    SRC_INDEX := 0,
                                    DEST_INDEX := 0,
                                    DEST => #row);
       RETURN;
   END_IF;

   #_status := MOVE_BLK_VARIANT(SRC := #row,
                                COUNT := 1,
                                SRC_INDEX := 0,
                                DEST_INDEX := 0,
                                DEST => #_string_row);
   #_string_row.cell_00.animation := #GRAY_BACKGROUND;
   #_string_row.cell_01.animation := #GRAY_BACKGROUND;
   #_status := MOVE_BLK_VARIANT(SRC := #_string_row,
                                COUNT := 1,
                                SRC_INDEX := 0,
                                DEST_INDEX := 0,
                                DEST => #row);
   RETURN;
END_FUNCTION

// folder: middleware

FUNCTION_BLOCK "Middleware"   // FB2, SCL
{ S7_Optimized_Access := 'TRUE' }
VERSION : 0.1
   VAR_IN_OUT
      database : "Database.UDT";
      hmi : "HMI_Interface.UDT";
      led : "LED_Interface.UDT";
   END_VAR
   VAR
      elements : "Elements";
      wires : "Wires";
   END_VAR
BEGIN
   #elements(database := #database.elements,
             hmi := #hmi.elements,
             led := #led.elements);

   #wires(database := #database.wires,
          hmi := #hmi.wires,
          led := #led.wires);
END_FUNCTION_BLOCK

// folder: wire

FUNCTION_BLOCK "Wire"   // FB1, SCL
{ S7_Optimized_Access := 'TRUE' }
VERSION : 0.1
   VAR_IN_OUT
      database : Real;
      hmi : "Row.(IOF.String_IOF.Real).UDT";
      led : "ADP.Row.2_Cells.UDT";
   END_VAR
BEGIN
   "Wire.Read"(database := #database,
               hmi := #hmi,
               led := #led);
END_FUNCTION_BLOCK

FUNCTION_BLOCK "Wires"   // FB4, SCL
{ S7_Optimized_Access := 'TRUE' }
VERSION : 0.1
   VAR_IN_OUT
      database : "Wires.Data.UDT";
      hmi : "Wires.HMI.UDT";
      led : "Wires.LED.UDT";
   END_VAR
   VAR
      aluminum : "Wire";
      calcium_silicon : "Wire";
      carbon : "Wire";
      custom : "Wire";
      heat : "Wire";
      sulfur : "Wire";
   END_VAR
BEGIN
   #aluminum(database := #database.aluminum,
             hmi := #hmi.aluminum,
             led := #led.aluminum);

   #calcium_silicon(database := #database.calcium_silicon,
                    hmi := #hmi.calcium_silicon,
                    led := #led.calcium_silicon);

   #carbon(database := #database.carbon,
           hmi := #hmi.carbon,
           led := #led.carbon);

   #custom(database := #database.custom,
           hmi := #hmi.custom,
           led := #led.custom);

   #heat(database := #database.heat,
         hmi := #hmi.heat,
         led := #led.heat);

   #sulfur(database := #database.sulfur,
           hmi := #hmi.sulfur,
           led := #led.sulfur);
END_FUNCTION_BLOCK

FUNCTION "Wire.Set" : Void   // FC1, SCL
{ S7_Optimized_Access := 'TRUE' }
VERSION : 0.1
BEGIN
END_FUNCTION

FUNCTION "Wire.Read" : Void   // FC2, SCL
{ S7_Optimized_Access := 'TRUE' }
VERSION : 0.1
   VAR_INPUT
      database : Real;
   END_VAR
   VAR_IN_OUT
      hmi : "Row.(IOF.String_IOF.Real).UDT";
      led : "ADP.Row.2_Cells.UDT";
   END_VAR
BEGIN
   "Wire.Read.HMI"(database := #database,
                   hmi := #hmi);
   "Wire.Read.LED"(database := #database,
                   led := #led);
END_FUNCTION

FUNCTION "Wire.Scale" : Real   // FC3, SCL
{ S7_Optimized_Access := 'TRUE' }
VERSION : 0.1
   VAR_INPUT
      value : Real;
   END_VAR
BEGIN
   #"Wire.Scale" := "Material.Scale"(#value);
END_FUNCTION

FUNCTION "Wire.Validate" : Void   // FC5, SCL
{ S7_Optimized_Access := 'TRUE' }
VERSION : 0.1
BEGIN
END_FUNCTION

FUNCTION "Wire.Animate" : Void   // FC7, SCL
{ S7_Optimized_Access := 'TRUE' }
VERSION : 0.1
   VAR_IN_OUT
      row : Bool;
   END_VAR
BEGIN
   "Material.Animate"(#row);
END_FUNCTION

FUNCTION "Wire.Read.HMI" : Void   // FC16, SCL
{ S7_Optimized_Access := 'TRUE' }
VERSION : 0.1
   VAR_INPUT
      database : Real;
   END_VAR
   VAR_IN_OUT
      hmi : "Row.(IOF.String_IOF.Real).UDT";
   END_VAR
BEGIN
   "Material.Read.HMI"(database := #database,
                       hmi := #hmi);
END_FUNCTION

FUNCTION "Wire.Read.LED" : Void   // FC17, SCL
{ S7_Optimized_Access := 'TRUE' }
VERSION : 0.1
   VAR_INPUT
      database : Real;
   END_VAR
   VAR_IN_OUT
      led : "ADP.Row.2_Cells.UDT";
   END_VAR
BEGIN
   "Material.Read.LED"(database := #database,
                       led := #led);
END_FUNCTION

// ===== library: MasterCopy "Copy of PLC data types in ADP Data" =====

// folder: ADP Data

TYPE "ADP: Encoded"
VERSION : 0.1
   STRUCT
      file_system : "ADP: Encoded: File System";
      formatting : "ADP: Encoded: Formatting";
   END_STRUCT;
END_TYPE

TYPE "ADP: Decoded"
   STRUCT
      color : "ADP: Decoded: Color";
      flash : "ADP: Decoded: Flash";
      horizontal_alignment : "ADP: Decoded: Horizontal Alignment";
      line_control : "ADP: Decoded: Line Control";
      scroll_speed : "ADP: Decoded: Scroll Speed";
      size_and_face : "ADP: Decoded: Size and Face";
      vertical_alignment : "ADP: Decoded: Vertical Alignment";
   END_STRUCT;
END_TYPE

TYPE "ADP: Decoded: Color"
   STRUCT
      black : String[8] := 'black';
      blue : String[8] := 'blue';
      green : String[8] := 'green';
      mix_1 : String[8] := 'mix 1';
      mix_2 : String[8] := 'mix 2';
      mix_3 : String[8] := 'mix 3';
      mix_4 : String[8] := 'mix 4';
      red : String[8] := 'red';
      white : String[8] := 'white';
      yellow : String[8] := 'yellow';
   END_STRUCT;
END_TYPE

TYPE "ADP: Decoded: Flash"
   STRUCT
      off : String[8] := 'off';
      on : String[8] := 'on';
   END_STRUCT;
END_TYPE

TYPE "ADP: Decoded: Horizontal Alignment"
   STRUCT
      center : String[8] := 'center';
      left : String[8] := 'left';
      right : String[8] := 'right';
   END_STRUCT;
END_TYPE

TYPE "ADP: Message Formats: Encoded"
   STRUCT
      color : String [5];
      flash : String [5];
      scroll_speed : String [5];
      size_and_face : String [5];
      vertical_alignment : String [5];
      horizontal_alignment : String [5];
   END_STRUCT;
END_TYPE

TYPE "ADP: Message Formats: Decoded"
   STRUCT
      color : String [20];
      flash : String [20];
      scroll_speed : String [20];
      size_and_face : String [20];
      vertical_alignment : String [20];
      horizontal_alignment : String [20];
   END_STRUCT;
END_TYPE

TYPE "ADP: Decoded: Scroll Speed"
   STRUCT
      slowest : String[9] := 'slowest';
      slow : String[9] := 'slow';
      normal : String[9] := 'normal';
      fast : String[9] := 'fast';
      fastest : String[9] := 'fastest';
   END_STRUCT;
END_TYPE

TYPE "ADP: Decoded: Size and Face"
   STRUCT
      bold_5 : String[11] := 'bold 5';
      bold_11 : String[11] := 'bold 11';
      bold_14 : String[11] := 'bold 14';
      bold_15 : String[11] := 'bold 15';
      bold_16 : String[11] := 'bold 16';
      bold_22 : String[11] := 'bold 22';
      bold_30 : String[11] := 'bold 30';
      bold_32 : String[11] := 'bold 32';
      bold_40 : String[11] := 'bold 40';
      normal_5 : String[11] := 'normal 5';
      normal_7 : String[11] := 'normal 7';
      normal_9 : String[11] := 'normal 9';
      normal_11 : String[11] := 'normal 11';
      normal_14 : String[11] := 'normal 14';
      normal_15 : String[11] := 'normal 15';
      normal_16 : String[11] := 'normal 16';
      normal_22 : String[11] := 'normal 22';
      normal_24 : String[11] := 'normal 24';
      normal_30 : String[11] := 'normal 30';
      normal_32 : String[11] := 'normal 32';
      normal_40 : String[11] := 'normal 40';
   END_STRUCT;
END_TYPE

TYPE "ADP: Decoded: Vertical Alignment"
   STRUCT
      bottom_hold : String[15] := 'bottom hold';
      fill_hold : String[15] := 'fill hold';
      middle_hold : String[15] := 'middle hold';
      top_hold : String[15] := 'top hold';
      bottom_scroll : String[15] := 'bottom scroll';
      fill_scroll : String[15] := 'fill scroll';
      middle_scroll : String[15] := 'middle scroll';
      top_scroll : String[15] := 'top scroll';
   END_STRUCT;
END_TYPE

TYPE "ADP: Encoded: File System"
   STRUCT
      "00 Start of Header" : String[5] := '$01';
      "01 Address" : String[5] := 'Z00';
      "02 Start of Text" : String[5] := '$02';
      "03 Command & File" : String[5] := 'AA';
      "04 END" : String[5] := '$04';
   END_STRUCT;
END_TYPE

TYPE "ADP: Encoded: Formatting"
   STRUCT
      color : "ADP: Encoded: Formatting: Color";
      flashing : "ADP: Encoded: Formatting: Flashing";
      horizontal_alignment : "ADP: Encoded: Formatting: Horizontal Alignment";
      line_control : "ADP: Encoded: Formatting: Line Control";
      scroll_speed : "ADP: Encoded: Formatting: Scroll Speed";
      size_and_face : "ADP: Encoded: Formatting: Size and Face";
      vertical_alignment : "ADP: Encoded: Formatting: Vertical Alignment";
   END_STRUCT;
END_TYPE

TYPE "ADP: Encoded: Formatting: Color"
   STRUCT
      black : String[5] := '$1C0';
      blue : String[5] := '$1C8';
      green : String[5] := '$1C2';
      mix_1 : String[5] := '$1C4';
      mix_2 : String[5] := '$1C5';
      mix_3 : String[5] := '$1C6';
      mix_4 : String[5] := '$1CY';
      red : String[5] := '$1C1';
      white : String[5] := '$1C9';
      yellow : String[5] := '$1C3';
   END_STRUCT;
END_TYPE

TYPE "ADP: Encoded: Formatting: Flashing"
   STRUCT
      off : String[5] := '$070';
      on : String[5] := '$071';
   END_STRUCT;
END_TYPE

TYPE "ADP: Encoded: Formatting: Size and Face"
   STRUCT
      bold_5 : String[5] := '$1AG';
      bold_11 : String[5] := '$1AH';
      bold_14 : String[5] := '$1A5';
      bold_15 : String[5] := '$1A6';
      bold_16 : String[5] := '$1A7';
      bold_22 : String[5] := '$1AC';
      bold_30 : String[5] := '$1AI';
      bold_32 : String[5] := '$1AJ';
      bold_40 : String[5] := '$1AK';
      normal_5 : String[5] := '$1A0';
      normal_7 : String[5] := '$1A1';
      normal_9 : String[5] := '$1A8';
      normal_11 : String[5] := '$1A9';
      normal_14 : String[5] := '$1A2';
      normal_15 : String[5] := '$1A3';
      normal_16 : String[5] := '$1A4';
      normal_22 : String[5] := '$1AA';
      normal_24 : String[5] := '$1AB';
      normal_30 : String[5] := '$1AD';
      normal_32 : String[5] := '$1AE';
      normal_40 : String[5] := '$1AF';
   END_STRUCT;
END_TYPE

TYPE "ADP: Encoded: Formatting: Horizontal Alignment"
   STRUCT
      center : String[5] := '$L1';
      left : String[5] := '$L0';
      right : String[5] := '$L2';
   END_STRUCT;
END_TYPE

TYPE "ADP: Encoded: Formatting: Vertical Alignment"
   STRUCT
      middle_hold : String[5] := '$1B b';
      fill_hold : String[5] := '$1B"b';
      bottom_hold : String[5] := '$1B&b';
      top_hold : String[5] := '$1B0b';
      bottom_scroll : String[5] := '$1B a';
      fill_scroll : String[5] := '$1B"a';
      middle_scroll : String[5] := '$1B&a';
      top_scroll : String[5] := '$1B0a';
   END_STRUCT;
END_TYPE

TYPE "ADP: Encoded: Formatting: Scroll Speed"
   STRUCT
      slowest : String[5] := '$15';
      slow : String[5] := '$16';
      normal : String[5] := '$17';
      fast : String[5] := '$18';
      fastest : String[5] := '$19';
   END_STRUCT;
END_TYPE

TYPE "ADP: Encoded: Formatting: Line Control"
   STRUCT
      new_line : String[5] := '$R';
      word_wrap : String[5] := '';
   END_STRUCT;
END_TYPE

TYPE "ADP: Decoded: Line Control"
   STRUCT
      new_line : String[9] := 'new line';
      word_wrap : String[9] := 'word wrap';
   END_STRUCT;
END_TYPE

(* ===== HMI "HMI_RT_1" =====
connection "HMI_Connection_1": ETHERNET, S7_1200_OMS

HMI tags "Default tag table"
   "Clock_Byte" : Byte = PLC Clock_Byte AT %MB0, 1 s
*)

(* ===== HMI "HMI_RT_1" =====

ScreenModuleEditorView "Row.IOF_IOF" 400x50
   IOField "I/O field_1" at 5,5 size 190x45; FormatPattern 9999999
   IOField "I/O field_2" at 200,5 size 195x45; FormatPattern 9999999
*)